{attribute 'GeneratedUsingTerminal: EL2252-0000-0016'}
{attribute addProperty BoxType "EL2252-0000-0016"}
{attribute addProperty Id "StartTimeAT %Q*ULINT8"}
{attribute addProperty CRC "3895366195"}
{attribute addProperty Size "8"}
TYPE DC_Sync_Start_E82E9233 EXTENDS OutputBase_10CEE7DE :
STRUCT
	{attribute addProperty Name "StartTime"}
	StartTime AT %Q* : ULINT;
END_STRUCT
END_TYPE

(* stored: Version 1.2.0.0, ProductVersion 3.1.4024.11
   DUT DC_Sync_Start_E82E9233: Id {e74f2124-d086-4f45-bd02-c19ea63fd1f0} *)
